INTERFACE I_Tagged EXTENDS I_Component

PROPERTY Tag : I_Tag
GET
END_GET
END_PROPERTY

END_INTERFACE

(* stored: Version 1.1.0.1
   Itf I_Tagged: Id {92a57a01-5096-46ab-961f-63d875b95829}
   Property Tag: Id {89260ffc-7430-48a1-b2e1-4c0eefce60ad}
   Get Get: Id {8e3bdc78-0098-46c9-9c83-30021dc1a8b2} *)
